FUNCTION_BLOCK Test_F_DINT_TO_UDINT_Conversion EXTENDS TUnitTestBase
VAR
    InputValue : DINT;
    ConvertedValue : UDINT;
END_VAR

InputValue := -20; // wrong sign
ConvertedValue := F_DINT_TO_UDINT(InputValue); // limit to zero

Assertion.AssertEquals_UDINT(
    Expected:= 0, 
    Actual:= ConvertedValue, 
    VariableName:= 'ConvertedValue');
    
TestFinished();

END_FUNCTION_BLOCK

(* stored: Version 1.1.0.1, ProductVersion 3.1.4024.4
   POU Test_F_DINT_TO_UDINT_Conversion: Id {4ca60ad8-5283-4117-a7ee-a2fae33f240a}, SpecialFunc None *)
